# EPICS StreamDevice protocol: protocols/sync_role.proto
Terminator = LF;
ExtraInput = Ignore;

set_sync_role {
	out "sync_role %s";
	in;
}

get_sync_role {
	out "sync_role";
	in "%s";
}
